// TIA Portal V19 export
FUNCTION "LAxisCtrlApcFr_ChangeCamOnTheFly_GetMasterCamData" : Void   // FC19508, LAD
{ S7_Optimized_Access := 'TRUE' }
// stored: IsIECCheckEnabled true, SetENOAutomatically true
   VAR_INPUT
      camUsed : TO_Cam;
      camFollowing : TO_Cam;
      axis : TO_SynchronousAxis;
   END_VAR
   VAR_OUTPUT
      effectiveMasterOffset : LReal;
      effectiveSlaveOffset : LReal;
      endLeadingValueCamUsed : LReal;
      startLeadingValueCamFollowing : LReal;
   END_VAR
BEGIN

REGION Network 1 (SCL)

   // Get offset
   #effectiveMasterOffset := #axis.StatusSynchronizedMotion.MasterOffset;
   #effectiveSlaveOffset := #axis.StatusSynchronizedMotion.SlaveOffset;
   #endLeadingValueCamUsed := #camUsed.StatusCam.EndLeadingValue;
   #startLeadingValueCamFollowing := #camFollowing.StatusCam.StartLeadingValue;
END_REGION
END_FUNCTION
